(* IEC 61131-3 sources: MXEN3002/deliverables/usb/st, 7 files *)

(* ---- FB_Actuator_T1.st ---- *)
(*
  FB_Actuator_T1  --  holdable double-solenoid actuator.
  Used for: Distributing swivel arm, Testing lift.

  Holdable = pause STOPS IT IMMEDIATELY mid-stroke (both valves off traps it in
  place); resume continues to the SAME target (no jerk home). Reset drives it
  directly home, aborting any stroke. Robust variant: a TON stall timer -- moving
  with the target sensor not reached within t_stall -- forces ERROR.

  States: 0 AT_HOME 1 TO_END 2 AT_END 3 TO_HOME 4 ERROR
  Milestone 1.5/1.6 (arm), 2.2/2.3 (lift). t_stall is an INPUT: tune in the lab.

  NOTE (milestone 1.9): this FB must NOT contain Station_2Y1/2Y2 (vacuum /
  ejector pulse). It drives only its own two solenoids. Vacuum lives in Main.
*)
FUNCTION_BLOCK FB_Actuator_T1
VAR_INPUT
    run_mode    : BOOL;
    pause_mode  : BOOL;
    reset_mode  : BOOL;
    error_mode  : BOOL;
    sensor_home : BOOL;          // at-home limit switch
    sensor_end  : BOOL;          // at-end  limit switch
    go          : BOOL;          // Main requests a stroke (hold TRUE = continuous)
    t_stall     : TIME := T#2s;  // stall timeout (lab-tunable)
    robust      : BOOL := FALSE; // TRUE enables stall detection (1.6 / 2.3)
END_VAR
VAR_OUTPUT
    at_home      : BOOL;
    to_end       : BOOL;
    at_end       : BOOL;
    to_home      : BOOL;
    valve_to_end : BOOL;         // Station_3Y2 (arm) / Station_1Y2 (lift up)
    valve_to_home: BOOL;         // Station_3Y1 (arm) / Station_1Y1 (lift down)
    error        : BOOL;
END_VAR
VAR
    state  : INT := 0;
    stall  : TON;
    moving : BOOL;
END_VAR

CASE state OF
0:  (* AT_HOME *)
    IF error_mode THEN state := 4;
    ELSIF reset_mode THEN
        IF NOT sensor_home THEN state := 3; END_IF;
    ELSIF run_mode AND go THEN
        state := 1;
    END_IF;
1:  (* TO_END *)
    IF error_mode THEN state := 4;
    ELSIF reset_mode THEN state := 3;          // abort stroke, go home
    ELSIF pause_mode THEN ;                     // freeze in place
    ELSIF sensor_end THEN state := 2;
    END_IF;
2:  (* AT_END *)
    IF error_mode THEN state := 4;
    ELSIF reset_mode THEN state := 3;
    ELSIF run_mode AND go THEN state := 3;      // continuous cycle
    END_IF;
3:  (* TO_HOME *)
    IF error_mode THEN state := 4;
    ELSIF pause_mode AND NOT reset_mode THEN ;  // freeze (reset overrides pause)
    ELSIF sensor_home THEN state := 0;
    END_IF;
4:  (* ERROR -- valves off, recover only via reset sequence *)
    IF reset_mode THEN
        IF sensor_home THEN state := 0; ELSE state := 3; END_IF;
    END_IF;
END_CASE;

// Valves derive from the final state; pause zeroes them (hold in place).
valve_to_end  := (state = 1) AND NOT pause_mode;
valve_to_home := (state = 3) AND NOT pause_mode;

// Stall detection: commanding a valve but not arriving.
moving := valve_to_end OR valve_to_home;
stall(IN := robust AND moving, PT := t_stall);
IF stall.Q THEN state := 4; END_IF;

IF state = 4 THEN
    valve_to_end := FALSE;
    valve_to_home := FALSE;
END_IF;

at_home := (state = 0);
to_end  := (state = 1);
at_end  := (state = 2);
to_home := (state = 3);
error   := (state = 4);

END_FUNCTION_BLOCK

(* ---- FB_Actuator_T2.st ---- *)
(*
  FB_Actuator_T2  --  stroke-completing single-acting cylinder, TWO limit sensors.
  Used for: Distributing ejection cylinder, Sorting branch 1 & branch 2.

  Stroke-completing = pause takes effect ONLY at end of stroke. If Stop is pressed
  mid-travel the cylinder finishes to the limit (extended or retracted) and halts
  there; it never stops mid-stroke. Single solenoid: valve ON = extend, valve OFF =
  spring retract. To halt extended in pause the valve is HELD on at AT_END.

  States: 0 AT_HOME(retracted) 1 TO_END(extend) 2 AT_END(extended) 3 TO_HOME(retract) 4 ERROR
  Milestone 1.7/1.8 (ejector), used again on Sorting branches (L.1). t_stall lab-tunable.
*)
FUNCTION_BLOCK FB_Actuator_T2
VAR_INPUT
    run_mode    : BOOL;
    pause_mode  : BOOL;
    reset_mode  : BOOL;
    error_mode  : BOOL;
    sensor_home : BOOL;          // retracted limit switch
    sensor_end  : BOOL;          // extended limit switch
    go          : BOOL;
    t_stall     : TIME := T#2s;
    robust      : BOOL := FALSE;
END_VAR
VAR_OUTPUT
    at_home      : BOOL;
    to_end       : BOOL;
    at_end       : BOOL;
    to_home      : BOOL;
    valve_extend : BOOL;
    error        : BOOL;
END_VAR
VAR
    state  : INT := 0;
    stall  : TON;
    moving : BOOL;
END_VAR

CASE state OF
0:  (* AT_HOME *)
    IF error_mode THEN state := 4;
    ELSIF reset_mode THEN
        IF NOT sensor_home THEN state := 3; END_IF;
    ELSIF run_mode AND go THEN state := 1;
    END_IF;
1:  (* TO_END -- stroke completes regardless of pause *)
    IF error_mode THEN state := 4;
    ELSIF sensor_end THEN state := 2;
    END_IF;
2:  (* AT_END -- valve held extended; only run advances to retract *)
    IF error_mode THEN state := 4;
    ELSIF reset_mode THEN state := 3;
    ELSIF run_mode THEN state := 3;
    END_IF;
3:  (* TO_HOME -- valve off, spring retracts, completes regardless of pause *)
    IF error_mode THEN state := 4;
    ELSIF sensor_home THEN state := 0;
    END_IF;
4:  (* ERROR *)
    IF reset_mode THEN
        IF sensor_home THEN state := 0; ELSE state := 3; END_IF;
    END_IF;
END_CASE;

valve_extend := (state = 1) OR (state = 2);
IF state = 4 THEN valve_extend := FALSE; END_IF;

moving := (state = 1) OR (state = 3);
stall(IN := robust AND moving, PT := t_stall);
IF stall.Q THEN
    state := 4;
    valve_extend := FALSE;
END_IF;

at_home := (state = 0);
to_end  := (state = 1);
at_end  := (state = 2);
to_home := (state = 3);
error   := (state = 4);

END_FUNCTION_BLOCK

(* ---- FB_Actuator_T3.st ---- *)
(*
  FB_Actuator_T3  --  stroke-completing single-acting cylinder, ONE limit sensor.
  Used for: Testing ejection cylinder (only a retracted switch, Station_2B1).

  Same contract as T2 but the EXTENDED end has no switch: it is inferred from a
  stroke timer (t_stroke). Because there is no extend sensor, stall is only
  detectable on the RETRACT leg (t_stall on failing to reach sensor_home). A
  cylinder held while extended is caught on the following retract attempt.
  Set t_stroke slightly longer than the real extend travel; tune in the lab.

  States: 0 AT_HOME 1 TO_END(timer) 2 AT_END 3 TO_HOME(sensor) 4 ERROR
  Milestone 2.4/2.5. Reused on Sorting stopper (single-sensor) per L.1.
*)
FUNCTION_BLOCK FB_Actuator_T3
VAR_INPUT
    run_mode    : BOOL;
    pause_mode  : BOOL;
    reset_mode  : BOOL;
    error_mode  : BOOL;
    sensor_home : BOOL;          // retracted limit switch (the only one)
    go          : BOOL;
    t_stroke    : TIME := T#1s;  // assumed extend time (no end sensor)
    t_stall     : TIME := T#2s;  // retract stall timeout
    robust      : BOOL := FALSE;
END_VAR
VAR_OUTPUT
    at_home      : BOOL;
    to_end       : BOOL;
    at_end       : BOOL;
    to_home      : BOOL;
    valve_extend : BOOL;
    error        : BOOL;
END_VAR
VAR
    state  : INT := 0;
    strokeT: TON;
    stallT : TON;
END_VAR

CASE state OF
0:  (* AT_HOME *)
    IF error_mode THEN state := 4;
    ELSIF reset_mode THEN
        IF NOT sensor_home THEN state := 3; END_IF;
    ELSIF run_mode AND go THEN state := 1;
    END_IF;
1:  (* TO_END -- no sensor, trust the stroke timer *)
    IF error_mode THEN state := 4;
    ELSIF strokeT.Q THEN state := 2;
    END_IF;
2:  (* AT_END *)
    IF error_mode THEN state := 4;
    ELSIF reset_mode THEN state := 3;
    ELSIF run_mode THEN state := 3;
    END_IF;
3:  (* TO_HOME -- retract, sensor_home ends it *)
    IF error_mode THEN state := 4;
    ELSIF sensor_home THEN state := 0;
    END_IF;
4:  (* ERROR *)
    IF reset_mode THEN
        IF sensor_home THEN state := 0; ELSE state := 3; END_IF;
    END_IF;
END_CASE;

valve_extend := (state = 1) OR (state = 2);
IF state = 4 THEN valve_extend := FALSE; END_IF;

strokeT(IN := (state = 1), PT := t_stroke);
stallT (IN := robust AND (state = 3), PT := t_stall);   // retract-only stall
IF stallT.Q THEN
    state := 4;
    valve_extend := FALSE;
END_IF;

at_home := (state = 0);
to_end  := (state = 1);
at_end  := (state = 2);
to_home := (state = 3);
error   := (state = 4);

END_FUNCTION_BLOCK

(* ---- FB_Panel.st ---- *)
(*
  FB_Panel  --  shared control-panel FSM for all three Festo stations.
  Implements milestone 1.4.

  States: 0=PAUSE (power-on) 1=RUN 2=RESET 3=ERROR
    PAUSE --S1--> RUN         RUN  --S2--> PAUSE
    PAUSE --S4--> RESET       RESET--S2 or reset_done--> PAUSE
    any --error_in--> ERROR   ERROR--S4--> RESET (error cleared, then homes)
  Invalid transitions (S1 in RESET, S4 in RUN, S1/S2 in ERROR) are ignored.
  Exactly one operational light (start/reset) is ever on.

  reset_done = "all actuators are home" (Main ANDs the FBs' at_home outputs).
  It lets RESET fall back to PAUSE once homing finishes, so error recovery is
  two operator presses (Reset then Start). In the panel-only milestone 1.4 there
  are no actuators, so tie reset_done := FALSE and RESET only exits on S2.
*)
FUNCTION_BLOCK FB_Panel
VAR_INPUT
    s1_start   : BOOL;   // Panel_S1  Start button
    s2_stop    : BOOL;   // Panel_S2  Stop button
    s4_reset   : BOOL;   // Panel_S4  Reset button
    error_in   : BOOL;   // latched fault from actuators / main control block
    reset_done : BOOL;   // TRUE when every actuator reports at_home
END_VAR
VAR_OUTPUT
    run_mode    : BOOL;
    reset_mode  : BOOL;
    pause_mode  : BOOL;
    error_mode  : BOOL;
    start_light : BOOL;  // Station_H1
    reset_light : BOOL;  // Station_H2
END_VAR
VAR
    state : INT := 0;    // 0 PAUSE (power-on default)
END_VAR

IF error_in AND state <> 3 THEN
    state := 3;                          // ERROR forced from any state
ELSIF state = 0 THEN                     // PAUSE
    IF s1_start THEN
        state := 1;
    ELSIF s4_reset THEN
        state := 2;
    END_IF;
ELSIF state = 1 THEN                     // RUN
    IF s2_stop THEN state := 0; END_IF;  // S4 ignored here
ELSIF state = 2 THEN                     // RESET
    IF s2_stop OR reset_done THEN state := 0; END_IF;   // S1 ignored here
ELSIF state = 3 THEN                     // ERROR
    IF s4_reset THEN state := 2; END_IF; // clears fault, begins reset/homing
END_IF;

run_mode    := (state = 1);
pause_mode  := (state = 0);
reset_mode  := (state = 2);
error_mode  := (state = 3);
start_light := run_mode;
reset_light := reset_mode;

END_FUNCTION_BLOCK

(* ---- Main_Distributing.st ---- *)
(*
  Main_Distributing  --  Station 1 top-level program (milestone 1.9 / 1.10).

  Blocks (milestone 1.9 asks for 4): FB_Panel, FB_Actuator_T1 (arm),
  FB_Actuator_T2 (ejector), and THIS Main. Main owns everything the FBs must
  not: the vacuum (Station_2Y1) and ejector-pulse (Station_2Y2) valves, the
  unused sensors (Station_B4 magazine-empty, IP_FI), the Q1/Q2 lights, the
  7-step cycle sequencer, and the 5-piece batch counter.

  Set ROBUST := FALSE to demo 1.9 (proper), TRUE to demo 1.10 (robust).
  The 7-step cycle mirrors milestone 1.9's numbered list exactly.
*)
PROGRAM Main_Distributing
VAR
    Panel   : FB_Panel;
    Arm     : FB_Actuator_T1;     // swivel arm  (home = magazine)
    Ejector : FB_Actuator_T2;     // magazine ejection cylinder
    si         : INT := 0;        // sequence step 0..6
    cycles     : INT := 0;        // workpieces completed this batch
    grip, drop : INT := 0;        // dwell counters for vacuum grip / drop
    go_arm, go_ej : BOOL;
    vacuum, eject_pulse : BOOL;
    fault, reset_done   : BOOL;
    ROBUST : BOOL := TRUE;        // 1.10 = TRUE, 1.9 = FALSE
    MAG    : INT  := 5;           // magazine capacity / batch size
END_VAR

reset_done := Arm.at_home AND Ejector.at_home;
Panel(s1_start := Panel_S1, s2_stop := Panel_S2, s4_reset := Panel_S4,
      error_in := fault, reset_done := reset_done);

IF Panel.reset_mode OR Panel.error_mode THEN
    si := 0; grip := 0; drop := 0; vacuum := FALSE; eject_pulse := FALSE;
    IF Panel.reset_mode THEN cycles := 0; END_IF;
END_IF;

go_arm := FALSE; go_ej := FALSE; eject_pulse := FALSE;
IF Panel.run_mode AND cycles < MAG THEN
    CASE si OF
    0:  go_arm := TRUE;  IF Arm.at_end  THEN si := 1; END_IF;   (* 1 arm downstream *)
    1:  go_ej  := TRUE;  IF Ejector.at_end  THEN si := 2; END_IF; (* 2 ejector push  *)
    2:  go_arm := TRUE;  IF Arm.at_home THEN si := 3; END_IF;   (* 3 arm upstream  *)
    3:  vacuum := TRUE;  grip := grip + 1;                       (* 4 vacuum grips  *)
        IF grip >= 1 THEN grip := 0; si := 4; END_IF;
    4:  go_ej := FALSE;  IF Ejector.at_home THEN si := 5; END_IF; (* 5 ejector retract *)
    5:  go_arm := TRUE;  IF Arm.at_end  THEN si := 6; END_IF;   (* 6 arm to end    *)
    6:  eject_pulse := TRUE; vacuum := FALSE; drop := drop + 1;  (* 7 drop + vac off *)
        IF drop >= 1 THEN drop := 0; cycles := cycles + 1; si := 0; END_IF;
    END_CASE;
END_IF;

Arm(run_mode := Panel.run_mode, pause_mode := Panel.pause_mode,
    reset_mode := Panel.reset_mode, error_mode := Panel.error_mode,
    sensor_home := Station_3S1, sensor_end := Station_3S2, go := go_arm,
    t_stall := T#2s, robust := ROBUST);

Ejector(run_mode := Panel.run_mode, pause_mode := Panel.pause_mode,
    reset_mode := Panel.reset_mode, error_mode := Panel.error_mode,
    sensor_home := Station_1B1, sensor_end := Station_1B2, go := go_ej,
    t_stall := T#2s, robust := ROBUST);

// Robust faults (1.10): stalled actuator, piece pulled off the vacuum
// (vacuum commanded but Station_2B1 gripped-sensor lost), or arm reaching the
// magazine with it empty (Station_B4).
fault := ROBUST AND ( Arm.error OR Ejector.error
    OR (Panel.run_mode AND vacuum AND NOT Station_2B1)
    OR (Panel.run_mode AND Arm.at_home AND Station_B4 AND si <> 0) );

// ---- physical outputs ----
Station_3Y2 := Arm.valve_to_end;       // Arm_to_Subsequent (downstream)
Station_3Y1 := Arm.valve_to_home;      // Arm_to_Magazine
Station_1Y1 := Ejector.valve_extend;   // Magazine_Eject
Station_2Y1 := vacuum      AND NOT Panel.error_mode;   // Vacuum_On
Station_2Y2 := eject_pulse AND NOT Panel.error_mode;   // Ejector_Pulse_On
Station_H1  := Panel.start_light;      // start light
Station_H2  := Panel.reset_light;      // reset light
Panel_H3    := (cycles >= MAG);        // Q1  batch of 5 complete
Panel_H4    := Panel.error_mode;       // Q2  error
// IP_FI (succeeding-station-free) is jumpered TRUE stand-alone; for the
// integrated line (L.2) gate step 6 delivery on IP_FI.

END_PROGRAM

(* ---- Main_Sorting.st ---- *)
(*
  Main_Sorting  --  Station 3 top-level program (milestone 3.1 / 3.2).

  Blocks (5): FB_Panel, FB_Actuator_T2 (branch 1), FB_Actuator_T2 (branch 2),
  FB_Actuator_T3 (stopper, single-acting timed release), and THIS Main. Main owns
  the conveyor (Station_K1), the sort decision, the three slide counters, the
  slide-full interlock and Q1/Q2.

  Classification:
    metal := Station_B2                 -> branch 1 (slide 1)
    red   := Station_B3 AND NOT Station_B2 (not black, not metal) -> branch 2 (slide 2)
    black := NOT Station_B3             -> straight through (slide 3)
  Any slide full (Station_B4 or a counter at cap) -> Q1 ON and station -> ERROR
  (test 3.1.2). Set ROBUST := FALSE for 3.1, TRUE for 3.2.
*)
PROGRAM Main_Sorting
VAR
    Panel   : FB_Panel;
    Branch1 : FB_Actuator_T2;
    Branch2 : FB_Actuator_T2;
    Stopper : FB_Actuator_T3;      // timed release, no limit switch
    pos     : INT := 0;            // conveyor position of the current piece 0..3
    dest    : INT := 0;            // 0 branch1  1 branch2  2 straight
    have    : BOOL;                // a piece is being routed
    s1c, s2c, s3c : INT := 0;      // slide counts (cap 5)
    conveyor, go_b1, go_b2, go_stop : BOOL;
    metal, red, black, slide_full : BOOL;
    fault, reset_done : BOOL;
    ROBUST : BOOL := TRUE;
    CAP    : INT  := 5;
END_VAR

reset_done := Branch1.at_home AND Branch2.at_home;
Panel(s1_start := Panel_S1, s2_stop := Panel_S2, s4_reset := Panel_S4,
      error_in := fault, reset_done := reset_done);

IF Panel.reset_mode OR Panel.error_mode THEN
    have := FALSE; pos := 0;
END_IF;

slide_full := Station_B4 OR (s1c >= CAP) OR (s2c >= CAP) OR (s3c >= CAP);

conveyor := FALSE; go_b1 := FALSE; go_b2 := FALSE; go_stop := FALSE;
IF Panel.run_mode AND NOT slide_full THEN
    IF NOT have THEN
        IF Part_AV THEN                        // classify newly released piece
            metal := Station_B2;
            black := NOT Station_B3;
            red   := Station_B3 AND NOT Station_B2;
            IF metal THEN dest := 0;
            ELSIF red THEN dest := 1;
            ELSE dest := 2; END_IF;
            have := TRUE; pos := 0;
            go_stop := TRUE;                   // pulse stopper to admit the piece
        END_IF;
    ELSE
        CASE dest OF
        0:  (* branch 1 *)
            IF pos < 1 THEN conveyor := TRUE; pos := pos + 1;
            ELSE
                go_b1 := TRUE;
                IF Branch1.at_end THEN s1c := s1c + 1; have := FALSE; END_IF;
            END_IF;
        1:  (* branch 2 *)
            IF pos < 2 THEN conveyor := TRUE; pos := pos + 1;
            ELSE
                go_b2 := TRUE;
                IF Branch2.at_end THEN s2c := s2c + 1; have := FALSE; END_IF;
            END_IF;
        2:  (* straight through to end slide *)
            IF pos < 3 THEN conveyor := TRUE; pos := pos + 1;
            ELSE s3c := s3c + 1; have := FALSE; END_IF;
        END_CASE;
    END_IF;
END_IF;

Branch1(run_mode := Panel.run_mode, pause_mode := Panel.pause_mode,
    reset_mode := Panel.reset_mode, error_mode := Panel.error_mode,
    sensor_home := Station_1B1, sensor_end := Station_1B2, go := go_b1,
    t_stall := T#2s, robust := ROBUST);

Branch2(run_mode := Panel.run_mode, pause_mode := Panel.pause_mode,
    reset_mode := Panel.reset_mode, error_mode := Panel.error_mode,
    sensor_home := Station_2B1, sensor_end := Station_2B2, go := go_b2,
    t_stall := T#2s, robust := ROBUST);

Stopper(run_mode := Panel.run_mode, pause_mode := Panel.pause_mode,
    reset_mode := Panel.reset_mode, error_mode := Panel.error_mode,
    sensor_home := TRUE, go := go_stop,
    t_stroke := T#1s, t_stall := T#2s, robust := ROBUST);

// Robust faults (3.2): a branch stalled/held, or any slide full. Piece-removed
// (a piece taken off the conveyor before a slide) is inferred as: routing a
// piece but Part_AV lost mid-line -- VERIFY sensor behaviour on the bench.
fault := (ROBUST AND (Branch1.error OR Branch2.error))
    OR (Panel.run_mode AND slide_full)
    OR (ROBUST AND Panel.run_mode AND have AND pos >= 1 AND NOT Part_AV);

// ---- physical outputs ----
Station_K1  := conveyor AND NOT Panel.error_mode;   // Conveyor Motor ON
Station_1Y1 := Branch1.valve_extend;                // Branch 1 extend
Station_2Y1 := Branch2.valve_extend;                // Branch 2 extend
Station_3Y1 := Stopper.valve_extend;                // Stopper retract (release)
Station_H1  := Panel.start_light;
Station_H2  := Panel.reset_light;
Station_H3  := slide_full;                          // Q1
Station_H4  := Panel.error_mode;                    // Q2
IP_N_FO     := Panel.run_mode;                      // station occupied

END_PROGRAM

(* ---- Main_Testing.st ---- *)
(*
  Main_Testing  --  Station 2 top-level program (milestone 2.6 / 2.7).

  Blocks (4): FB_Panel, FB_Actuator_T1 (lift, REUSED from Station 1),
  FB_Actuator_T3 (ejector, single retract sensor), and THIS Main. Main owns the
  colour/height sort logic, the blower (Station_3Y1), the top/bottom slide
  counters, the safety-beam interlock, and Q1/Q2.

  Piece classification from sensors:
    black   := NOT Station_B2         (B2 = "workpiece not black")
    tall    := Station_B5             (height correct = tall = red/metal)
    white   = not black AND not tall   -> bottom slide
    red/metal = not black AND tall     -> top slide (blower 1 s)
    black                              -> bottom slide, no lift

  Beam polarity: Station_B4 is a through-beam (TRUE = clear). beam_blocked below
  is NOT Station_B4 -- VERIFY this polarity on the real bench and flip if needed.
  Set ROBUST := FALSE for 2.6, TRUE for 2.7.
*)
PROGRAM Main_Testing
VAR
    Panel   : FB_Panel;
    Lift    : FB_Actuator_T1;      // home = down, end = up
    Ejector : FB_Actuator_T3;      // single retract sensor
    ps      : INT := 0;            // 0 IDLE 1 LIFTING 2 HEIGHT 3 EJECT_TOP
                                   // 4 EJECT_BOTTOM 5 LOWER
    dest_bottom : BOOL;            // current piece routes to bottom after lower
    bottom, top : INT := 0;        // slide counts (cap 5)
    beam_ctr    : INT := 0;        // safety-beam block duration (scans)
    go_lift, go_ej, blower : BOOL;
    black, tall, beam_blocked : BOOL;
    fault, reset_done, beam_fault, proc_fault : BOOL;
    ROBUST : BOOL := TRUE;
    CAP    : INT  := 5;
    BEAM_LIMIT : INT := 3;         // scans (~3 s) before beam -> error
END_VAR

reset_done := Lift.at_home AND Ejector.at_home;
Panel(s1_start := Panel_S1, s2_stop := Panel_S2, s4_reset := Panel_S4,
      error_in := fault, reset_done := reset_done);

IF Panel.reset_mode OR Panel.error_mode THEN
    ps := 0; beam_ctr := 0; proc_fault := FALSE; dest_bottom := FALSE;
END_IF;

beam_blocked := NOT Station_B4;
beam_fault := FALSE;
IF beam_blocked AND (ps = 1 OR ps = 5) THEN
    beam_ctr := beam_ctr + 1;
    IF ROBUST AND beam_ctr >= BEAM_LIMIT THEN beam_fault := TRUE; END_IF;
ELSIF NOT beam_blocked THEN
    beam_ctr := 0;
END_IF;

go_lift := FALSE; go_ej := FALSE; blower := FALSE;
IF Panel.run_mode THEN
    CASE ps OF
    0:  (* IDLE: latch class of the presented workpiece *)
        IF Part_AV THEN
            black := NOT Station_B2;
            IF black THEN ps := 4;              // straight to bottom, no lift
            ELSE ps := 1; END_IF;
        END_IF;
    1:  (* LIFTING to the height sensor *)
        IF NOT beam_blocked THEN
            go_lift := TRUE;
            IF Lift.at_end THEN ps := 2; END_IF;
        END_IF;
    2:  (* HEIGHT decision *)
        tall := Station_B5;
        IF tall THEN                            // red / metal -> top slide
            IF top < CAP THEN ps := 3; ELSE ps := 5; dest_bottom := FALSE; END_IF;
        ELSE                                    // white -> bottom slide
            IF ROBUST AND bottom >= CAP THEN
                proc_fault := TRUE;             // bottom full: stop at entry, error
            ELSE
                dest_bottom := TRUE; ps := 5;
            END_IF;
        END_IF;
    3:  (* EJECT to TOP slide, blower on *)
        go_ej := TRUE; blower := TRUE;
        IF Ejector.at_end THEN top := top + 1; dest_bottom := FALSE; ps := 5; END_IF;
    4:  (* EJECT to BOTTOM slide *)
        go_ej := TRUE;
        IF Ejector.at_end THEN bottom := bottom + 1; ps := 0; END_IF;
    5:  (* LOWER lift home, then dispatch *)
        go_lift := TRUE;
        IF Lift.at_home THEN
            IF dest_bottom THEN ps := 4; ELSE ps := 0; END_IF;
        END_IF;
    END_CASE;
END_IF;

Lift(run_mode := Panel.run_mode, pause_mode := Panel.pause_mode,
    reset_mode := Panel.reset_mode, error_mode := Panel.error_mode,
    sensor_home := Station_1B2, sensor_end := Station_1B1, go := go_lift,
    t_stall := T#2s, robust := ROBUST);

Ejector(run_mode := Panel.run_mode, pause_mode := Panel.pause_mode,
    reset_mode := Panel.reset_mode, error_mode := Panel.error_mode,
    sensor_home := Station_2B1, go := go_ej,
    t_stroke := T#1s, t_stall := T#2s, robust := ROBUST);

fault := ROBUST AND (Lift.error OR Ejector.error OR beam_fault OR proc_fault);

// ---- physical outputs ----
Station_1Y1 := Lift.valve_to_home;     // Lift Down
Station_1Y2 := Lift.valve_to_end;      // Lift Up
Station_2Y1 := Ejector.valve_extend;   // Advance Ejecting Cylinder
Station_3Y1 := blower AND NOT Panel.error_mode;  // Air Cushion (blower, ~1 s)
Station_H1  := Panel.start_light;
Station_H2  := Panel.reset_light;
Station_H3  := (bottom >= CAP);        // Q1  bottom slide full
Station_H4  := Panel.error_mode;       // Q2
IP_N_FO     := Panel.run_mode;         // station occupied (integrated line)

END_PROGRAM
